// Returns the datatype of a variable as a string using its pointer and size.
// Variables allocated in dynamic memory are not supported.
FUNCTION FsF_GetTypeName : FsT_Str
VAR_INPUT
	Variable : ANY;
END_VAR
VAR 
	nTmp : UDINT := SIZEOF(FsF_GetTypeName);
END_VAR

_FsGVL.fbTcComIecApplicationInfo
	.GetInterface()
	.GetDatatypeNameByAddress(TO_UDINT(Variable.diSize), Variable.pValue, nTmp, ADR(FsF_GetTypeName));

END_FUNCTION

(* stored: Version 1.1.0.1, ProductVersion 3.1.4024.4
   POU FsF_GetTypeName: Id {272394df-f52a-4096-af79-4769dfbdb581}, SpecialFunc None *)
